// TIA Portal V20 export
ORGANIZATION_BLOCK "Main"   // OB127, LAD, ProgramCycle
TITLE = "Main Program Sweep (Cycle)"
// stored: IsIECCheckEnabled true, Namespace C3, SetENOAutomatically false
   VAR_INPUT
      Initial_Call : Bool;   // Initial call of this OB
      Remanence : Bool;   // =True, if remanent data are available
   END_VAR
BEGIN

REGION Network 1
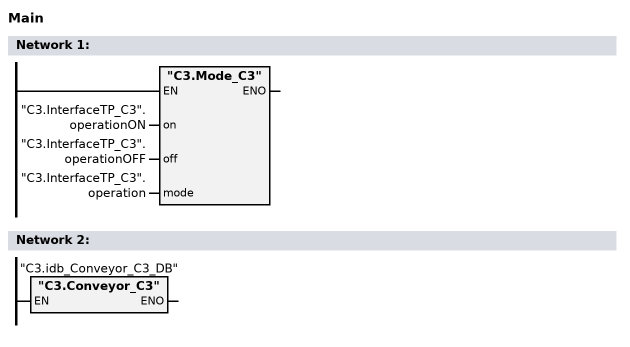
   RUNG wire#powerrail
      "C3.Mode_C3"(on := "C3.InterfaceTP_C3".operationON, off := "C3.InterfaceTP_C3".operationOFF, mode := "C3.InterfaceTP_C3".operation)
   END_RUNG
   // the same network as SCL:
   "C3.Mode_C3"(on := "C3.InterfaceTP_C3".operationON,
                off := "C3.InterfaceTP_C3".operationOFF,
                mode := "C3.InterfaceTP_C3".operation);
END_REGION

REGION Network 2
   RUNG wire#powerrail
      "C3.idb_Conveyor_C3_DB"()
   END_RUNG
   // the same network as SCL:
   "C3.idb_Conveyor_C3_DB"();   // "C3.Conveyor_C3"
END_REGION
END_ORGANIZATION_BLOCK
